Staubli VAL3: onF1Event.pgx

program onF1Event()
  local bool l_bYes
  local string l_sMessage
  local string l_sItem
  local string l_sButton[2]
  local string l_sPage
  local InstrItem l_iItem
begin
  // look if the bButton is enable
  if bButton[0]
    //
    //
    // the SIMULATION is disable when cycle is active
    //
    if !cycleStatus:bCycle and find(left(sEvent,5),"-")==-1
      call language:message(l_sMessage,214)
      // get the yes_no button Key
      call language:getYesNo(l_sButton)
      // ask the question
      call use:yes_no(l_sMessage,l_sButton,l_bYes)
      if l_bYes
        call prog:getItem(l_iItem,nIndex)
        cycleStatus:iToSuperV=l_iItem
        cycleStatus:nInterfaceToSV=3
        logMsg("[KERNEL] INTERFACE:Simulation of the item: "+sEvent)
        wait(cycleStatus:nInterfaceToSV==-1)
        // load the production page
        l_sPage="simulation"
        call loadPage("kernel/page/production",l_sPage)
        call use:setView(false)
      endIf
    endIf
  endIf
end
